FUNCTION StringAssembly : STRING

VAR_IN_OUT
	liste : ARRAY [*] OF WORD; 
END_VAR

VAR
	counter : INT;
END_VAR

END_FUNCTION

(* stored: Version 1.1.0.1, ProductVersion 3.1.4024.12
   POU POU: Id {2641f0bf-5dd4-4550-a3f0-60310d82f2c8}, SpecialFunc None *)
